(* Logix 5000 project; controller MOVE Emulate 5570 rev 36.11; software revision 36.00 *)

TASK MainTask (continuous, watchdog 500 ms) : MainProgram, Model

MODULES
   Local : Emulate 5570 (ICP 2, rev 36.11)
       : 1756-IB16 (ICP 3, rev 3.1, Input RPI 20 ms)
       : vendor 1 type 7 code 16 (ICP 4, rev 3.1, Output RPI 20 ms)
END_MODULES

ADD_ON_INSTRUCTION Emulate   (* revision 1.0 *)
VAR_INPUT
   EmSELSW : DINT; {required}
END_VAR
VAR_OUTPUT
   SW0 : BOOL; {required}
   SW1 : BOOL; {required}
   SW2 : BOOL; {access Read Only, required}
END_VAR

ROUTINE Logic   (* ladder *)
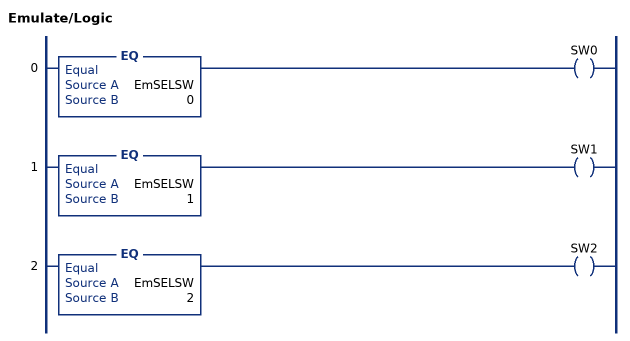
   0: EQ(EmSELSW,0)OTE(SW0);
   1: EQ(EmSELSW,1)OTE(SW1);
   2: EQ(EmSELSW,2)OTE(SW2);
END_ROUTINE
END_ADD_ON_INSTRUCTION

VAR_GLOBAL   (* controller tags *)
   OUTPUT : ALIAS FOR Local:4:O.Data.0;   // Process Output
   SEL_SW_1 : ALIAS FOR Local:3:I.Data.0;   // Selector Switch, Position 1
   SEL_SW_2 : ALIAS FOR Local:3:I.Data.1;   // Selector Switch, Position 2
   SEL_SW_3 : ALIAS FOR Local:3:I.Data.2;   // Selector Switch, Position 3
   START : ALIAS FOR Local:3:I.Data.14;   // START Momentary N.O. Pushbutton
END_VAR

PROGRAM MainProgram   (* main routine MainRoutine *)
VAR
   DWELL : TIMER := (PRE := 15000);   // Process Timer
        .EN   // Process Timer Enabled
        .ACC   // Process Timer Accumulated
        .PRE   // Process Timer Preset
        .DN   // Process Timer Complete
   HMI_ACC : REAL;   // Operator Panel Timer Accumulated
   HMI_ENABLE_DISABLE : BOOL;   // Allows Hardwired Panel
   HMI_PB : INT := 2;   // Operator Panel Pushbuttons
   HMI_PB_1 : BOOL;   // Operator Panel Pushbutton 1
   HMI_PB_2 : BOOL;   // Operator Panel Pushbutton 2
   HMI_PB_3 : BOOL;   // Operator Panel Pushbutton 3
   HMI_PRE : REAL;   // Operator Panel Timer Preset
   ONE_SHOT : SINT[1];   // One Shot Control Array
   PRE_SET_1 : INT := 10000;   // Preset No. 1
   PRE_SET_2 : INT := 15000;   // Preset No. 2
   PRE_SET_3 : INT := 20000;   // Preset No. 3
END_VAR

ROUTINE HMI_ROUTINE   (* ladder *)
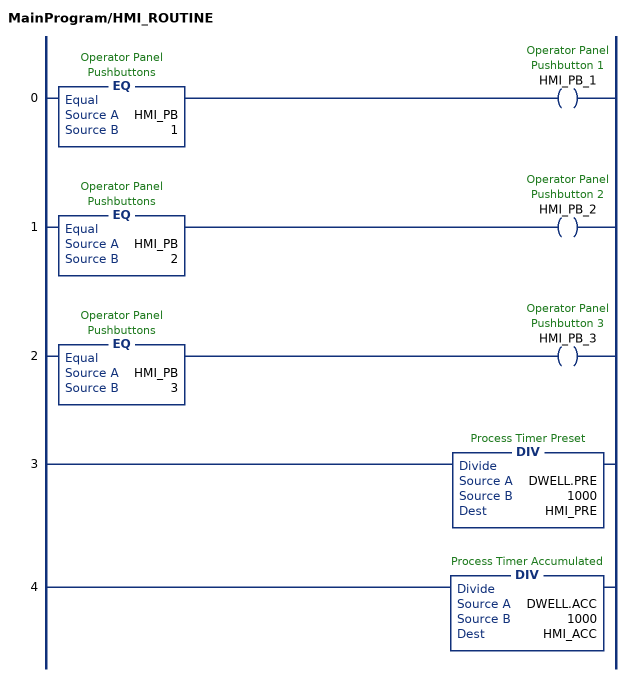
   0: EQ(HMI_PB,1)OTE(HMI_PB_1);
   1: EQ(HMI_PB,2)OTE(HMI_PB_2);
   2: EQ(HMI_PB,3)OTE(HMI_PB_3);
   3: DIV(DWELL.PRE,1000,HMI_PRE);
   4: DIV(DWELL.ACC,1000,HMI_ACC);
END_ROUTINE

ROUTINE MainRoutine   (* ladder *)
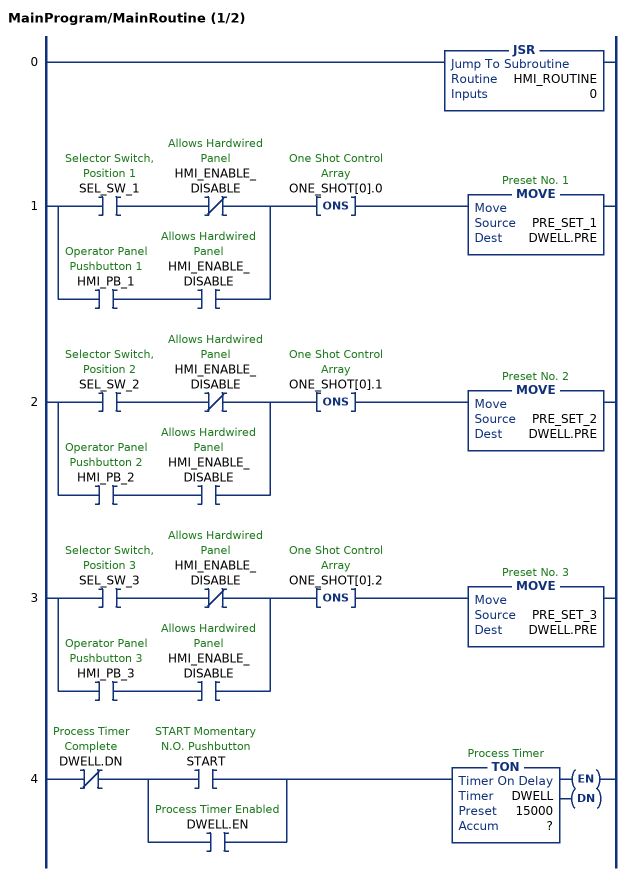
   0: JSR(HMI_ROUTINE,0);
   1: [XIC(SEL_SW_1) XIO(HMI_ENABLE_DISABLE) ,XIC(HMI_PB_1) XIC(HMI_ENABLE_DISABLE) ]ONS(ONE_SHOT[0].0)MOVE(PRE_SET_1,DWELL.PRE);
   2: [XIC(SEL_SW_2) XIO(HMI_ENABLE_DISABLE) ,XIC(HMI_PB_2) XIC(HMI_ENABLE_DISABLE) ]ONS(ONE_SHOT[0].1)MOVE(PRE_SET_2,DWELL.PRE);
   3: [XIC(SEL_SW_3) XIO(HMI_ENABLE_DISABLE) ,XIC(HMI_PB_3) XIC(HMI_ENABLE_DISABLE) ]ONS(ONE_SHOT[0].2)MOVE(PRE_SET_3,DWELL.PRE);
   4: XIO(DWELL.DN)[XIC(START) ,XIC(DWELL.EN) ]TON(DWELL,?,?);
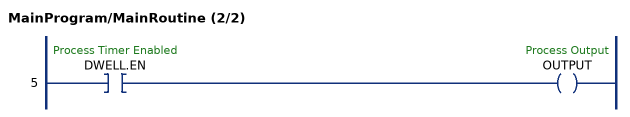
   5: XIC(DWELL.EN)OTE(OUTPUT);
END_ROUTINE
END_PROGRAM

PROGRAM Model   (* main routine Emulate *)
VAR
   emSELSW : DINT;
   emSW : Emulate := (SW0 := 1);
END_VAR

ROUTINE Emulate   (* ladder *)
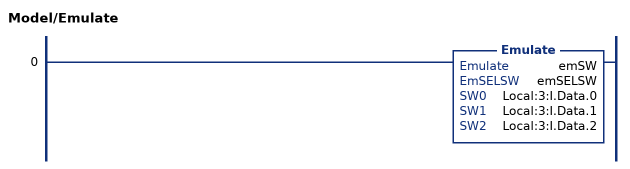
   0: Emulate(emSW,emSELSW,Local:3:I.Data.0,Local:3:I.Data.1,Local:3:I.Data.2);
END_ROUTINE
END_PROGRAM
